// TIA Portal V20 export
TYPE "LWONIK_typeFromSafetyEstopStatus"
// stored: Access Published
   STRUCT
      mainOpEmoPressed : Bool;   // EMO Pressed
      unwinderCenterEmoPressed : Bool;   // EMO Pressed
      jrOutPutEmoPressed : Bool;   // EMO Pressed
      pHmiEmoPressed : Bool;   // EMO Pressed
      ba10EmoPressed : Bool;   // EMO Pressed
      ba15EmoPressed : Bool;   // EMO Pressed
      ba40EmoPressed : Bool;   // EMO Pressed
      ba60EmoPressed : Bool;   // EMO Pressed
   END_STRUCT;
END_TYPE
